PROGRAM pouMcWarnings
VAR
	
idbMsgWarn: FB_CheckMessageBounds;
END_VAR

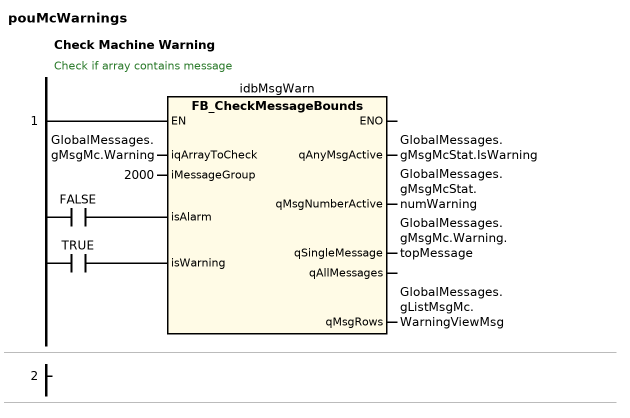
// NETWORK 1: Check Machine Warning
// Check if array contains message
idbMsgWarn(
    iqArrayToCheck := GlobalMessages.gMsgMc.Warning,
    iMessageGroup := 2000,
    isAlarm := FALSE,
    isWarning := TRUE,
    qAnyMsgActive => GlobalMessages.gMsgMcStat.IsWarning,
    qMsgNumberActive => GlobalMessages.gMsgMcStat.numWarning,
    qSingleMessage => GlobalMessages.gMsgMc.Warning.topMessage,
    qMsgRows => GlobalMessages.gListMsgMc.WarningViewMsg); // FB_CheckMessageBounds

// NETWORK 2

END_PROGRAM

(* stored: Version 1.1.0.1, ProductVersion 3.1.4024.12
   POU pouMcWarnings: Id {e2069892-172e-4d15-8119-82e0ee3317a8}, SpecialFunc None *)
